Fanuc KAREL source: kd00048.KL

-- PROVISIONAL review KL for V940-1; original PC SHA256 dc846656b1bc4ab57c9fca785251b092990a7953b18d00dabbfa1a4c63ea6e0d
-- Incomplete behavior may be omitted. Consult companion uncertainty JSON. Do not deploy.
PROGRAM KD00048
%NOLOCKGROUP
BEGIN
  -- V9_ZERO_TABLE_METADATA_HINT layout=0001; no indexed target words; source/name/runtime held
  -- UNRESOLVED_PC offsets 5-29; opcodes 01,22,1C,9D,2C,08,82,0B
  -- UNRESOLVED_PC offsets 34-38; opcodes 7F
END KD00048
